PROGRAM MAIN_Cutter
VAR
	State: INT;
	Start: INT;
	FuncDelay : Delay;	
END_VAR

IF GVL_Kitchen.System_Start = 0 THEN
 	FuncDelay;
	ELSE	
		CASE State OF
		0: 
			IF GVL_kitchen.Food_Cut < 2 THEN
				FuncDelay;
				GVL_Kitchen.Food_Cut := GVL_Kitchen.Food_Cut +1;
				ELSE 
					state := 1;
			END_IF;
		1:
			IF GVL_kitchen.Food_Spiced < 2 THEN
				GVL_Kitchen.Food_Cut := GVL_Kitchen.Food_Cut -1;
				FuncDelay;
				GVL_Kitchen.Food_Spiced := GVL_Kitchen.Food_Spiced +1;
				ELSE 
					state := 2;
			END_IF;
		2:
			IF GVL_kitchen.Food_Cooked > 0 THEN
			GVL_Kitchen.Food_Cooked := GVL_Kitchen.Food_Cooked -1;
			FuncDelay;
			GVL_Kitchen.Food_Plated := GVL_Kitchen.Food_Plated +1;
			ELSE 
				state := 0;
			END_IF;
		
		END_CASE
END_IF

END_PROGRAM

(* stored: Version 1.1.0.1, ProductVersion 3.1.4024.15
   POU MAIN_Cutter: Id {f1df099b-19f3-47d0-858e-fbde7c1af039}, SpecialFunc None *)
